// TIA Portal V20 export
TYPE "LER_TypeFATModeInterface"
// stored: Access Published
   STRUCT
      ModeSelect { S7_SetPoint := 'True'} : "LER_TypeFATMode_ModeSelect";
      HoursTest : Struct
         ProcessValue { S7_SetPoint := 'True'} : "LER_TypeFATMode_HoursTest_ProcessValue";
         SetValue { S7_SetPoint := 'True'} : "LER_TypeFATMode_HoursTest_SetValue";
      END_STRUCT;
      Capability : Struct
         ProcessValue { S7_SetPoint := 'True'} : "LER_TypeFATMode_Capability_ProcessValue";
         SetValue { S7_SetPoint := 'True'} : "LER_TypeFATMode_Capability_SetValue";
      END_STRUCT;
      Sampling : Struct
         ProcessValue { S7_SetPoint := 'True'} : "LER_TypeFATMode_Sampling_ProcessValue";
         SetValue { S7_SetPoint := 'True'} : "LER_TypeFATMode_Sampling_SetValue";
      END_STRUCT;
   END_STRUCT;
END_TYPE
